(* CODESYS project SPT_NC_Axis.library
   Company: Beckhoff Automation LLC
   DefaultNamespace: SPT_NCAxis
   Version: 3.0.3
   Placeholder: SPT NC Axis
   Title: SPT NC Axis

Project tree, tasks and I/O mapping:
  libraries: SPT Base Types, * (Beckhoff Automation LLC); SPT Drives, * (Beckhoff Automation LLC); SPT NC Homing, * (Beckhoff Automation LLC); Tc2_MC2, * (Beckhoff Automation GmbH); Tc2_System, * (Beckhoff Automation GmbH); Tc3_Module, * (Beckhoff Automation GmbH)
  Function Blocks/
    function block FB_BasicAxis [ST]: Disable, Enable, Home, Jog, MoveAbsolute, MoveModulo, MoveRelative, MoveVelocity, Reset, Stop, WriteBoolParameter, WriteParameter, Acceleration, Deceleration, Jerk, Velocity, ActualAcceleration, ActualPosition, ActualPositionModulo, ActualTorque, ActualVelocity, PositionLag, SetAcceleration, SetPosition, SetPositionModulo, SetVelocity, Enabled, InPosition, Stopped, Axis, HomeMethod, Override, ResetMethod, CyclicLogic, CallFBs, Initialize, AxisParameters
    function block FB_RingBuffer_MCMoveAbsolute [ST]: CurrentFB, GetNewFB
    function block FB_RingBuffer_MCMoveModulo [ST]: CurrentFB, GetNewFB
    function block FB_RingBuffer_MCMoveRelative [ST]: CurrentFB, GetNewFB
    function block FB_RingBuffer_MCMoveVelocity [ST]: CurrentFB, GetNewFB
  Interfaces/
    interface I_BasicAxis: Disable, Enable, Home, Jog, MoveAbsolute, MoveModulo, MoveRelative, MoveVelocity, Reset, Stop, WriteBoolParameter, WriteParameter, Acceleration, Deceleration, Jerk, Velocity, ActualAcceleration, ActualPosition, ActualPositionModulo, ActualTorque, ActualVelocity, PositionLag, SetAcceleration, SetPosition, SetPositionModulo, SetVelocity, Enabled, InPosition, Stopped, Axis, HomeMethod, Override, ResetMethod
    interface I_MotionSequence: Axis, Execute
  Project Information/
    function F_GetCompany [ST]
    function F_GetTitle [ST]
    function F_GetVersion [ST]
  Version/
    global variables Global_Version
  global variables Parameters_NCAxis
*)

// Version/Global_Version
{attribute 'TcGenerated'}
{attribute 'no-analysis'}
{attribute 'linkalways'}
// This function has been automatically generated from the project information.
VAR_GLOBAL CONSTANT
	{attribute 'const_non_replaced'}
	stLibVersion_SPT_NC_Axis : ST_LibVersion := (iMajor := 3, iMinor := 0, iBuild := 3, iRevision := 0, nFlags := 1, sVersion := '3.0.3');
END_VAR

// Parameters_NCAxis
{attribute 'qualified_only'}
VAR_GLOBAL CONSTANT
    ALLOW_UNLINKED_NC_AXES : BOOL := FALSE;
END_VAR

// Function Blocks/FB_BasicAxis
FUNCTION_BLOCK FB_BasicAxis EXTENDS FB_CyclicFB IMPLEMENTS I_BasicAxis
VAR
    _Axis           : AXIS_REF;
    _Velocity       : LREAL;
    _Acceleration   : LREAL;
    _Deceleration   : LREAL;
    _Jerk           : LREAL;
    ipHomeMethod    : I_MotionSequence;
    ipResetMethod   : I_MotionSequence;
    _AxisParameters : ST_AxisParameterSet;
END_VAR

VAR
    MCPower                   : MC_Power;
    RingBuffer_MCMoveAbsolute : FB_RingBuffer_MCMoveAbsolute;
    RingBuffer_MCMoveRelative : FB_RingBuffer_MCMoveRelative;
    RingBuffer_MCMoveVelocity : FB_RingBuffer_MCMoveVelocity;
    RingBuffer_MCMoveModulo   : FB_RingBuffer_MCMoveModulo;
    MCMoveAbsolute            : POINTER TO MC_MoveAbsolute;
    MCMoveRelative            : POINTER TO MC_MoveRelative;
    MCMoveVelocity            : POINTER TO MC_MoveVelocity;
    MCMoveModulo              : POINTER TO MC_MoveModulo;
    MCJog                     : MC_Jog;
    MCHalt                    : MC_Halt;
    DefaultHome               : FB_HomeRoutine_SetZeroHere;
    DefaultReset              : FB_ResetRoutine_CoEDrive;
    MCReadParameterSet        : MC_ReadParameterSet;
    MCWriteParameter          : MC_WriteParameterPersistent;
    MCWriteBoolParameter      : MC_WriteBoolParameterPersistent;
    HomePreviouslyErrored     : BOOL;
    ResetPreviouslyErrored    : BOOL;
END_VAR

//There should be no code in the function block body

METHOD Disable : BOOL
IF _Busy THEN
    RETURN;
END_IF

MCPower(Axis            := _Axis,
        Enable          := FALSE,
        Enable_Positive := FALSE,
        Enable_Negative := FALSE);

Disable := TRUE;
END_METHOD

METHOD Enable : BOOL
IF _Busy OR _Error THEN
    RETURN;
END_IF

MCPower(Axis            := _Axis,
        Enable          := TRUE,
        Enable_Positive := TRUE,
        Enable_Negative := TRUE);

Enable := TRUE;
END_METHOD

METHOD Home : BOOL
IF _Busy OR _Error OR ipHomeMethod = 0 THEN
    RETURN;
END_IF

//This is used to trap circular errors (I_MotionStratery resets error bit on next execute)
HomePreviouslyErrored := FALSE;
ipHomeMethod.Execute();
Home := TRUE;
END_METHOD

METHOD Jog : BOOL
VAR_INPUT
    JogFW    : BOOL;
    JogBW    : BOOL;
    JogMode  : E_JogMode;
    Position : LREAL;
END_VAR
IF _Error THEN
    RETURN;
END_IF

MCJog(Axis         := _Axis,
      JogForward   := JogFW,
      JogBackwards := JogBW,
      Mode         := JogMode,
      Position     := Position,
      Velocity     := _Velocity,
      Acceleration := _Acceleration,
      Deceleration := _Deceleration,
      Jerk         := _Jerk);
END_METHOD

METHOD MoveAbsolute : BOOL
VAR_INPUT
    Position      : LREAL;
    AbortPrevious : BOOL;
END_VAR
IF _Error THEN
    RETURN;
ELSE
    IF (_Busy AND NOT AbortPrevious) THEN
        RETURN;
    END_IF
END_IF

MCMoveAbsolute := RingBuffer_MCMoveAbsolute.GetNewFB();
MCMoveAbsolute^(Axis         := _Axis,
                Execute      := TRUE,
                Position     := Position,
                Velocity     := _Velocity,
                Acceleration := _Acceleration,
                Deceleration := _Deceleration,
                Jerk         := _Jerk);

MoveAbsolute := TRUE;
END_METHOD

METHOD MoveModulo : BOOL
VAR_INPUT
    Position      : LREAL;
    Direction     : MC_Direction;
    AbortPrevious : BOOL;
END_VAR
IF _Error THEN
    RETURN;
ELSE
    IF (_Busy AND NOT AbortPrevious) THEN
        RETURN;
    END_IF
END_IF

MCMoveModulo := RingBuffer_MCMoveModulo.GetNewFB();
MCMoveModulo^(Axis         := _Axis,
              Execute      := TRUE,
              Position     := Position,
              Velocity     := _Velocity,
              Acceleration := _Acceleration,
              Deceleration := _Deceleration,
              Jerk         := _Jerk,
              Direction    := Direction);

MoveModulo := TRUE;
END_METHOD

METHOD MoveRelative : BOOL
VAR_INPUT
    Distance      : LREAL;
    AbortPrevious : BOOL;
END_VAR
IF _Error THEN
    RETURN;
ELSE
    IF (_Busy AND NOT AbortPrevious) THEN
        RETURN;
    END_IF
END_IF

MCMoveRelative := RingBuffer_MCMoveRelative.GetNewFB();
MCMoveRelative^(Axis         := _Axis,
                Execute      := TRUE,
                Distance     := Distance,
                Velocity     := _Velocity,
                Acceleration := _Acceleration,
                Deceleration := _Deceleration,
                Jerk         := _Jerk);

MoveRelative := TRUE;
END_METHOD

METHOD MoveVelocity : BOOL
VAR_INPUT
    Velocity      : LREAL;
    AbortPrevious : BOOL;
END_VAR
IF _Error THEN
    RETURN;
ELSE
    IF (_Busy AND NOT AbortPrevious) THEN
        RETURN;
    END_IF
END_IF

IF ABS(Velocity) > _AxisParameters.fVeloMaximum THEN
    Trace('Velocity setpoint exceeds axis limit');
ELSIF Velocity = 0 THEN
    Trace('Velocity setpoint is 0; this will not work');
END_IF

IF Velocity = 0 THEN
    RETURN;
ELSIF Velocity < 0 THEN
    MCMoveVelocity            := RingBuffer_MCMoveVelocity.GetNewFB();
    MCMoveVelocity^.Direction := MC_Negative_Direction;
ELSE
    MCMoveVelocity            := RingBuffer_MCMoveVelocity.GetNewFB();
    MCMoveVelocity^.Direction := MC_Positive_Direction;
END_IF

_Velocity := ABS(Velocity);
MCMoveVelocity^(Axis         := _Axis,
                Execute      := TRUE,
                Velocity     := Velocity,
                Acceleration := _Acceleration,
                Deceleration := _Deceleration,
                Jerk         := _Jerk);

MoveVelocity := TRUE;
END_METHOD

METHOD Reset : BOOL
IF _Busy OR ipResetMethod = 0 THEN
    RETURN;
END_IF

//This is used to trap circular errors (I_MotionStratery resets error bit on next execute)
ResetPreviouslyErrored := FALSE;
IF ipResetMethod.Execute() THEN
    IF MCMoveAbsolute <> 0 THEN
        IF MCMoveAbsolute^.Error THEN
            MCMoveAbsolute^(Axis := _Axis, Execute := FALSE);
        END_IF
    END_IF

    IF MCMoveRelative <> 0 THEN
        IF MCMoveRelative^.Error THEN
            MCMoveRelative^(Axis := _Axis, Execute := FALSE);
        END_IF
    END_IF

    IF MCMoveVelocity <> 0 THEN
        IF MCMoveVelocity^.Error THEN
            MCMoveVelocity^(Axis := _Axis, Execute := FALSE);
        END_IF
    END_IF

    IF MCMoveModulo <> 0 THEN
        IF MCMoveModulo^.Error THEN
            MCMoveModulo^(Axis := _Axis, Execute := FALSE);
        END_IF
    END_IF

    IF MCHalt.Error THEN
        MCHalt(Axis := _Axis, Execute := FALSE);
    END_IF

    IF MCReadParameterSet.Error THEN
        MCReadParameterSet(Axis := _Axis, Parameter := _AxisParameters, Execute := FALSE);
    END_IF

    IF MCWriteBoolParameter.Error THEN
        MCWriteBoolParameter(Axis := _Axis, Execute := FALSE);
    END_IF

    IF MCWriteParameter.Error THEN
        MCWriteParameter(Axis := _Axis, Execute := FALSE);
    END_IF

    _Error   := FALSE;
    _ErrorID := 0;
    Reset    := TRUE;
END_IF
END_METHOD

METHOD Stop : BOOL
IF _Error AND _Axis.Status.Error THEN
    (* It's possible that a function block errored but
	not the NC itself--in this case we can allow a stop command.
	If the NC axis has a real fault then we want a successful reset first *)
    RETURN;
END_IF

MCHalt(Axis         := _Axis,
       Execute      := TRUE,
       Deceleration := _Deceleration,
       Jerk         := _Jerk);

Stop := TRUE;
END_METHOD

METHOD WriteBoolParameter : BOOL
VAR_INPUT
    ParameterNumber : MC_AxisParameter;
    Value           : BOOL;
END_VAR
IF _Busy OR _Error THEN
    RETURN;
END_IF

MCWriteBoolParameter(Axis            := _Axis,
                     Execute         := TRUE,
                     ParameterNumber := ParameterNumber,
                     Value           := Value);

WriteBoolParameter := TRUE;
END_METHOD

METHOD WriteParameter : BOOL
VAR_INPUT
    ParameterNumber : MC_AxisParameter;
    Value           : LREAL;
END_VAR
IF _Busy OR _Error THEN
    RETURN;
END_IF

MCWriteParameter(Axis            := _Axis,
                 Execute         := TRUE,
                 ParameterNumber := ParameterNumber,
                 Value           := Value);

WriteParameter := TRUE;
END_METHOD

PROPERTY Acceleration : LREAL
GET
Acceleration := _Acceleration;
END_GET
SET
IF Acceleration > _AxisParameters.fAccelerationMax THEN
    Trace('Acceleration setpoint exceeds axis limit');
END_IF

_Acceleration := Acceleration;
END_SET
END_PROPERTY

PROPERTY Deceleration : LREAL
GET
Deceleration := _Deceleration;
END_GET
SET
IF Deceleration > _AxisParameters.fDecelerationMax THEN
    Trace('Deceleration setpoint exceeds axis limit');
END_IF

_Deceleration := Deceleration;
END_SET
END_PROPERTY

PROPERTY Jerk : LREAL
GET
Jerk := _Jerk;
END_GET
SET
_Jerk := Jerk;
END_SET
END_PROPERTY

PROPERTY Velocity : LREAL
GET
Velocity := _Velocity;
END_GET
SET
IF Velocity > _AxisParameters.fVeloMaximum THEN
    Trace('Velocity setpoint exceeds axis limit');
END_IF

_Velocity := Velocity;
END_SET
END_PROPERTY

PROPERTY ActualAcceleration : LREAL
GET
ActualAcceleration := Axis.NcToPlc.ActAcc;
END_GET
END_PROPERTY

PROPERTY ActualPosition : LREAL
GET
ActualPosition := Axis.NcToPlc.ActPos;
END_GET
END_PROPERTY

PROPERTY ActualPositionModulo : LREAL
GET
ActualPositionModulo := Axis.NcToPlc.ModuloActPos;
END_GET
END_PROPERTY

PROPERTY ActualTorque : LREAL
GET
ActualTorque := Axis.NcToPlc.ActTorque;
END_GET
END_PROPERTY

PROPERTY ActualVelocity : LREAL
GET
ActualVelocity := Axis.NcToPlc.ActVelo;
END_GET
END_PROPERTY

PROPERTY PositionLag : LREAL
GET
PositionLag := Axis.NcToPlc.PosDiff;
END_GET
END_PROPERTY

PROPERTY SetAcceleration : LREAL
GET
SetAcceleration := Axis.NcToPlc.SetAcc;
END_GET
END_PROPERTY

PROPERTY SetPosition : LREAL
GET
SetPosition := Axis.NcToPlc.SetPos;
END_GET
END_PROPERTY

PROPERTY SetPositionModulo : LREAL
GET
SetPositionModulo := Axis.NcToPlc.ModuloSetPos;
END_GET
END_PROPERTY

PROPERTY SetVelocity : LREAL
GET
SetVelocity := Axis.NcToPlc.SetVelo;
END_GET
END_PROPERTY

PROPERTY Enabled : BOOL
GET
Enabled := MCPower.Status;
END_GET
END_PROPERTY

PROPERTY InPosition : BOOL
GET
InPosition := _Axis.Status.InTargetPosition;
END_GET
END_PROPERTY

PROPERTY Stopped : BOOL
GET
Stopped := _Axis.Status.NotMoving OR _Axis.Status.Disabled;
END_GET
END_PROPERTY

PROPERTY Axis : REFERENCE TO AXIS_REF
GET
Axis REF= _Axis;
END_GET
END_PROPERTY

PROPERTY HomeMethod : I_MotionSequence
GET
HomeMethod := ipHomeMethod;
END_GET
SET
ipHomeMethod      := HomeMethod;
ipHomeMethod.Axis := THIS^;
END_SET
END_PROPERTY

PROPERTY Override : LREAL
GET
Override := MCPower.Override;
END_GET
SET
IF Override >= 0 AND Override <= 100 THEN
    MCPower.Override := Override;
END_IF
END_SET
END_PROPERTY

PROPERTY ResetMethod : I_MotionSequence
GET
ResetMethod := ipResetMethod;
END_GET
SET
ipResetMethod      := ResetMethod;
ipResetMethod.Axis := THIS^;
END_SET
END_PROPERTY

METHOD PUBLIC CyclicLogic
VAR_INPUT
END_VAR
IF NOT _InitComplete THEN
    _InitComplete := THIS^.Initialize();
    RETURN;
END_IF

//Call local FBs
THIS^.CallFBs();
END_METHOD

METHOD PROTECTED CallFBs : BOOL
_Axis.ReadStatus();

(* MC_Power *)
MCPower(Axis := _Axis);
IF MCPower.Error THEN
    _Error   := TRUE;
    _ErrorID := MCPower.ErrorID;
END_IF

(* MC_MoveAbsolute *)
RingBuffer_MCMoveAbsolute(Axis := _Axis);
IF (MCMoveAbsolute <> 0) AND_THEN NOT MCMoveAbsolute^.Busy THEN
    IF MCMoveAbsolute^.Error THEN
        _Error   := TRUE;
        _ErrorID := MCMoveAbsolute^.ErrorID;
    ELSE
        MCMoveAbsolute^(Axis := _Axis, Execute := FALSE);
    END_IF
END_IF

(* MC_MoveRelative *)
RingBuffer_MCMoveRelative(Axis := _Axis);
IF (MCMoveRelative <> 0) AND_THEN NOT MCMoveRelative^.Busy THEN
    IF MCMoveRelative^.Error THEN
        _Error   := TRUE;
        _ErrorID := MCMoveRelative^.ErrorID;
    ELSE
        MCMoveRelative^(Axis := _Axis, Execute := FALSE);
    END_IF
END_IF

(* MC_MoveVelocity *)
RingBuffer_MCMoveVelocity(Axis := _Axis);
IF (MCMoveVelocity <> 0) AND_THEN NOT MCMoveVelocity^.Busy THEN
    IF MCMoveVelocity^.Error THEN
        _Error   := TRUE;
        _ErrorID := MCMoveVelocity^.ErrorID;
    ELSE
        MCMoveVelocity^(Axis := _Axis, Execute := FALSE);
    END_IF
END_IF

(* MC_MoveModulo *)
RingBuffer_MCMoveModulo(Axis := _Axis);
IF (MCMoveModulo <> 0) AND_THEN NOT MCMoveModulo^.Busy THEN
    IF MCMoveModulo^.Error THEN
        _Error   := TRUE;
        _ErrorID := MCMoveModulo^.ErrorID;
    ELSE
        MCMoveModulo^(Axis := _Axis, Execute := FALSE);
    END_IF
END_IF

(*MC_Jog*)
MCJog(Axis := _Axis);
IF MCJog.Error THEN
    _Error   := TRUE;
    _ErrorID := MCJog.ErrorID;
END_IF

(* MC_MoveHalt *)
MCHalt(Axis := _Axis);
IF NOT MCHalt.Busy THEN
    IF MCHalt.Error THEN
        _Error   := TRUE;
        _ErrorID := MCHalt.ErrorID;
    ELSE
        MCHalt(Axis := _Axis, Execute := FALSE);
    END_IF
END_IF

(* FB_HomeRoutine_SetZeroHere *)
IF ipHomeMethod <> 0 AND_THEN ipHomeMethod.Axis <> 0 THEN
    ipHomeMethod.CyclicLogic();
    IF NOT ipHomeMethod.Busy THEN
        IF ipHomeMethod.Error AND NOT HomePreviouslyErrored THEN
            //This is used to trap circular errors (I_MotionStratery resets error bit on next execute)
            HomePreviouslyErrored := TRUE;
            _Error                := TRUE;
            _ErrorID              := ipHomeMethod.ErrorID;
        END_IF
    END_IF
END_IF

(* FB_ResetRoutine_CoEDrive *)
IF ipResetMethod <> 0 AND_THEN ipResetMethod.Axis <> 0 THEN
    ipResetMethod.CyclicLogic();
    IF NOT ipResetMethod.Busy AND NOT ResetPreviouslyErrored THEN
        IF ipResetMethod.Error THEN
            //This is used to trap circular errors (I_MotionStratery resets error bit on next execute)
            ResetPreviouslyErrored := TRUE;
            _Error                 := TRUE;
            _ErrorID               := ipResetMethod.ErrorID;
        END_IF
    END_IF
END_IF

(* MC_WriteParameterPersistent *)
MCWriteParameter(Axis := _Axis);
IF NOT MCWriteParameter.Busy THEN
    IF MCWriteParameter.Error THEN
        _Error   := TRUE;
        _ErrorID := MCWriteParameter.ErrorID;
    ELSE
        MCWriteParameter(Axis := _Axis, Execute := FALSE);
    END_IF
END_IF

(* MC_WriteBoolParameterPersistent *)
MCWriteBoolParameter(Axis := _Axis);
IF NOT MCWriteBoolParameter.Busy THEN
    IF MCWriteBoolParameter.Error THEN
        _Error   := TRUE;
        _ErrorID := MCWriteBoolParameter.ErrorID;
    ELSE
        MCWriteBoolParameter(Axis := _Axis, Execute := FALSE);
    END_IF
END_IF

_Busy := ((MCMoveAbsolute <> 0) AND_THEN MCMoveAbsolute^.Busy) OR ((MCMoveRelative <> 0) AND_THEN MCMoveRelative^.Busy) OR ((MCMoveVelocity <> 0) AND_THEN MCMoveVelocity^.Busy) OR
         ((MCMoveModulo <> 0) AND_THEN MCMoveModulo^.Busy) OR MCJog.Busy OR MCHalt.Busy OR ((ipHomeMethod <> 0) AND_THEN ipHomeMethod.Busy) OR ((ipResetMethod <> 0) AND_THEN ipResetMethod.Busy) OR
         MCWriteParameter.Busy OR MCWriteBoolParameter.Busy;
END_METHOD

METHOD PROTECTED Initialize : BOOL
VAR_INST
    LinkMissing : BOOL;
END_VAR
// Verify that the AXIS_REF is actually linked with the NC
IF F_GetMappingStatus(ADR(_Axis.NcToPlc), SIZEOF(_Axis.NcToPlc)) <> EPlcMappingStatus.MS_Mapped THEN
    IF NOT Parameters_NCAxis.ALLOW_UNLINKED_NC_AXES THEN
        IF NOT LinkMissing THEN
            Trace('Axis is not linked to NC');
            LinkMissing := TRUE;
        END_IF

        RETURN;
    END_IF
END_IF

IF F_GetMappingStatus(ADR(_Axis.PlcToNc), SIZEOF(_Axis.PlcToNc)) <> EPlcMappingStatus.MS_Mapped THEN
    IF NOT Parameters_NCAxis.ALLOW_UNLINKED_NC_AXES THEN
        IF NOT LinkMissing THEN
            Trace('Axis is not linked to NC');
            LinkMissing := TRUE;
        END_IF

        RETURN;
    END_IF
END_IF

// AxisId will be populated by the NC when it finishes starting

// This prevents requesting motion before NC Init/nuisance errors
IF _Axis.NcToPlc.AxisId = 0 THEN
    IF NOT Parameters_NCAxis.ALLOW_UNLINKED_NC_AXES THEN
        RETURN;
    END_IF
END_IF

// Use default home and reset methods until they are set by parent
IF ipHomeMethod = 0 THEN
    THIS^.HomeMethod := DefaultHome;
END_IF

IF ipResetMethod = 0 THEN
    THIS^.ResetMethod := DefaultReset;
END_IF

// Read all NC parameters
IF Parameters_NCAxis.ALLOW_UNLINKED_NC_AXES THEN
    Initialize := TRUE;
ELSE
    MCReadParameterSet(Parameter := _AxisParameters, Axis := _Axis, Execute := TRUE);
    IF NOT MCReadParameterSet.Busy THEN
        IF MCReadParameterSet.Error THEN
            _Error   := TRUE;
            _ErrorID := MCReadParameterSet.ErrorID;
        ELSIF MCReadParameterSet.Done THEN
            _Velocity     := _AxisParameters.fVeloSlowManual;
            _Acceleration := _AxisParameters.fAcceleration;
            _Deceleration := _AxisParameters.fDeceleration;
            _Jerk         := _AxisParameters.fJerk;
            Trace('Axis initialization complete');
            Initialize := TRUE;
        END_IF

        MCReadParameterSet(Parameter := _AxisParameters, Axis := _Axis, Execute := FALSE);
    END_IF
END_IF
END_METHOD

PROPERTY AxisParameters : REFERENCE TO ST_AxisParameterSet
GET
AxisParameters REF= _AxisParameters;
END_GET
END_PROPERTY

END_FUNCTION_BLOCK

// Interfaces/I_BasicAxis
INTERFACE I_BasicAxis EXTENDS I_CyclicFB

METHOD PUBLIC Disable : BOOL
VAR_INPUT
END_VAR
END_METHOD

METHOD PUBLIC Enable : BOOL
VAR_INPUT
END_VAR
END_METHOD

METHOD PUBLIC Home : BOOL
VAR_INPUT
END_VAR
END_METHOD

METHOD Jog : BOOL
VAR_INPUT
    JogFW    : BOOL;
    JogBW    : BOOL;
    JogMode  : E_JogMode;
    Position : LREAL;
END_VAR
END_METHOD

METHOD PUBLIC MoveAbsolute : BOOL
VAR_INPUT
    Position      : LREAL;
    AbortPrevious : BOOL;
END_VAR
END_METHOD

METHOD MoveModulo : BOOL
VAR_INPUT
    Position      : LREAL;
    Direction     : MC_Direction;
    AbortPrevious : BOOL;
END_VAR
END_METHOD

METHOD PUBLIC MoveRelative : BOOL
VAR_INPUT
    Distance      : LREAL;
    AbortPrevious : BOOL;
END_VAR
END_METHOD

METHOD MoveVelocity : BOOL
VAR_INPUT
    Velocity      : LREAL;
    AbortPrevious : BOOL;
END_VAR
END_METHOD

METHOD PUBLIC Reset : BOOL
END_METHOD

METHOD Stop : BOOL
END_METHOD

METHOD WriteBoolParameter : BOOL
VAR_INPUT
    ParameterNumber : MC_AxisParameter;
    Value           : BOOL;
END_VAR
END_METHOD

METHOD WriteParameter : BOOL
VAR_INPUT
    ParameterNumber : MC_AxisParameter;
    Value           : LREAL;
END_VAR
END_METHOD

PROPERTY Acceleration : LREAL
GET
END_GET
SET
END_SET
END_PROPERTY

PROPERTY Deceleration : LREAL
GET
END_GET
SET
END_SET
END_PROPERTY

PROPERTY Jerk : LREAL
GET
END_GET
SET
END_SET
END_PROPERTY

PROPERTY Velocity : LREAL
GET
END_GET
SET
END_SET
END_PROPERTY

PROPERTY ActualAcceleration : LREAL
GET
END_GET
END_PROPERTY

PROPERTY ActualPosition : LREAL
GET
END_GET
END_PROPERTY

PROPERTY ActualPositionModulo : LREAL
GET
END_GET
END_PROPERTY

PROPERTY ActualTorque : LREAL
GET
END_GET
END_PROPERTY

PROPERTY ActualVelocity : LREAL
GET
END_GET
END_PROPERTY

PROPERTY PositionLag : LREAL
GET
END_GET
END_PROPERTY

PROPERTY SetAcceleration : LREAL
GET
END_GET
END_PROPERTY

PROPERTY SetPosition : LREAL
GET
END_GET
END_PROPERTY

PROPERTY SetPositionModulo : LREAL
GET
END_GET
END_PROPERTY

PROPERTY SetVelocity : LREAL
GET
END_GET
END_PROPERTY

PROPERTY Enabled : BOOL
GET
END_GET
END_PROPERTY

PROPERTY InPosition : BOOL
GET
END_GET
END_PROPERTY

PROPERTY Stopped : BOOL
GET
END_GET
END_PROPERTY

PROPERTY Axis : REFERENCE TO AXIS_REF
GET
END_GET
END_PROPERTY

PROPERTY HomeMethod : I_MotionSequence
SET
END_SET
END_PROPERTY

PROPERTY Override : LREAL
GET
END_GET
SET
END_SET
END_PROPERTY

PROPERTY ResetMethod : I_MotionSequence
SET
END_SET
END_PROPERTY

END_INTERFACE

// Interfaces/I_MotionSequence
INTERFACE I_MotionSequence EXTENDS I_CyclicFB

PROPERTY Axis : I_BasicAxis
GET
END_GET
SET
END_SET
END_PROPERTY

METHOD Execute : BOOL
END_METHOD

END_INTERFACE

// Function Blocks/FB_RingBuffer_MCMoveAbsolute
FUNCTION_BLOCK FB_RingBuffer_MCMoveAbsolute
VAR_IN_OUT
    Axis : AXIS_REF;
END_VAR

VAR_OUTPUT
END_VAR

VAR
    MCMoveAbsoluteCA : ARRAY[0..1] OF MC_MoveAbsolute;
    _CurrentFB       : UDINT;
    i                : UDINT;
END_VAR

(* This buffer ensures you always have a clean FB to use for a move *)

FOR i := 0 TO 1 DO
    MCMoveAbsoluteCA[i](Axis := Axis);
END_FOR

PROPERTY CurrentFB : POINTER TO MC_MoveAbsolute
GET
CurrentFB := ADR(MCMoveAbsoluteCA[_CurrentFB]);
END_GET
END_PROPERTY

METHOD GetNewFB : POINTER TO MC_MoveAbsolute
VAR_INPUT
END_VAR
_CurrentFB := _CurrentFB + 1;
IF _CurrentFB > 1 THEN
    MCMoveAbsoluteCA[1].Execute := FALSE;
    _CurrentFB                  := 0;
ELSE
    MCMoveAbsoluteCA[_CurrentFB - 1].Execute := FALSE;
END_IF

GetNewFB := ADR(MCMoveAbsoluteCA[_CurrentFB]);
END_METHOD

END_FUNCTION_BLOCK

// Function Blocks/FB_RingBuffer_MCMoveRelative
FUNCTION_BLOCK FB_RingBuffer_MCMoveRelative
VAR_IN_OUT
    Axis : AXIS_REF;
END_VAR

VAR_OUTPUT
END_VAR

VAR
    MCMoveRelative : ARRAY[0..1] OF MC_MoveRelative;
    _CurrentFB     : UDINT;
    i              : UDINT;
END_VAR

(* This buffer ensures you always have a clean FB to use for a move *)

FOR i := 0 TO 1 DO
    MCMoveRelative[i](Axis := Axis);
END_FOR

PROPERTY CurrentFB : POINTER TO MC_MoveRelative
GET
CurrentFB := ADR(MCMoveRelative[_CurrentFB]);
END_GET
END_PROPERTY

METHOD GetNewFB : POINTER TO MC_MoveAbsolute
VAR_INPUT
END_VAR
_CurrentFB := _CurrentFB + 1;
IF _CurrentFB > 1 THEN
    MCMoveRelative[1].Execute := FALSE;
    _CurrentFB                := 0;
ELSE
    MCMoveRelative[_CurrentFB - 1].Execute := FALSE;
END_IF

GetNewFB := ADR(MCMoveRelative[_CurrentFB]);
END_METHOD

END_FUNCTION_BLOCK

// Function Blocks/FB_RingBuffer_MCMoveVelocity
FUNCTION_BLOCK FB_RingBuffer_MCMoveVelocity
VAR_IN_OUT
    Axis : AXIS_REF;
END_VAR

VAR_OUTPUT
END_VAR

VAR
    MCMoveVelocity : ARRAY[0..1] OF MC_MoveVelocity;
    _CurrentFB     : UDINT;
    i              : UDINT;
END_VAR

(* This buffer ensures you always have a clean FB to use for a move *)

FOR i := 0 TO 1 DO
    MCMoveVelocity[i](Axis := Axis);
END_FOR

PROPERTY CurrentFB : POINTER TO MC_MoveVelocity
GET
CurrentFB := ADR(MCMoveVelocity[_CurrentFB]);
END_GET
END_PROPERTY

METHOD GetNewFB : POINTER TO MC_MoveAbsolute
VAR_INPUT
END_VAR
_CurrentFB := _CurrentFB + 1;
IF _CurrentFB > 1 THEN
    MCMoveVelocity[1].Execute := FALSE;
    _CurrentFB                := 0;
ELSE
    MCMoveVelocity[_CurrentFB - 1].Execute := FALSE;
END_IF

GetNewFB := ADR(MCMoveVelocity[_CurrentFB]);
END_METHOD

END_FUNCTION_BLOCK

// Function Blocks/FB_RingBuffer_MCMoveModulo
FUNCTION_BLOCK FB_RingBuffer_MCMoveModulo
VAR_IN_OUT
    Axis : AXIS_REF;
END_VAR

VAR_OUTPUT
END_VAR

VAR
    MCMoveModulo : ARRAY[0..1] OF MC_MoveModulo;
    _CurrentFB   : UDINT;
    i            : UDINT;
END_VAR

(* This buffer ensures you always have a clean FB to use for a move *)

FOR i := 0 TO 1 DO
    MCMoveModulo[i](Axis := Axis);
END_FOR

PROPERTY CurrentFB : POINTER TO MC_MoveModulo
GET
CurrentFB := ADR(MCMoveModulo[_CurrentFB]);
END_GET
END_PROPERTY

METHOD GetNewFB : POINTER TO MC_MoveAbsolute
VAR_INPUT
END_VAR
_CurrentFB := _CurrentFB + 1;
IF _CurrentFB > 1 THEN
    MCMoveModulo[1].Execute := FALSE;
    _CurrentFB              := 0;
ELSE
    MCMoveModulo[_CurrentFB - 1].Execute := FALSE;
END_IF

GetNewFB := ADR(MCMoveModulo[_CurrentFB]);
END_METHOD

END_FUNCTION_BLOCK

// Project Information/F_GetCompany
// This function has been automatically generated from the project information.
{attribute 'signature_flag' := '1073741824'}
{attribute 'TcGenerated'}
{attribute 'no-analysis'}
FUNCTION F_GetCompany : WSTRING
VAR_INPUT
	
END_VAR

F_GetCompany := "Beckhoff Automation LLC";

END_FUNCTION

// Project Information/F_GetTitle
// This function has been automatically generated from the project information.
{attribute 'signature_flag' := '1073741824'}
{attribute 'TcGenerated'}
{attribute 'no-analysis'}
FUNCTION F_GetTitle : WSTRING
VAR_INPUT
	
END_VAR

F_GetTitle := "SPT NC Axis";

END_FUNCTION

// Project Information/F_GetVersion
// This function has been automatically generated from the project information.
{attribute 'signature_flag' := '1073741824'}
{attribute 'TcGenerated'}
{attribute 'no-analysis'}
FUNCTION F_GetVersion : ST_LibVersion
VAR_INPUT
	
END_VAR

F_GetVersion.iMajor := 3;
F_GetVersion.iMinor := 0;
F_GetVersion.iBuild := 3;
F_GetVersion.iRevision := 0;
F_GetVersion.sVersion := '3.0.3';
F_GetVersion.nFlags := 1;

END_FUNCTION
